TYPE ERROR_MESSAGE : WSTRING(2000); END_TYPE

(* stored: Version 1.1.0.1
   DUT ERROR_MESSAGE: Id {8739ee3e-8f85-4784-a1cf-58d690d8f414} *)
